# EPICS autosave request: autosave/pu610k.req
#
# List of PVs to autosave.  Assume $(BASE) is the detector base PV,
# $(CHAN) is the channel number/name, and $(IOC) is the IOC base PV.
#
$(BASE):$(CHAN):ENABLE_RBV
$(BASE):$(CHAN):VOLTAGE
$(BASE):$(CHAN):CHARGE_INHIBIT
$(BASE):AUTO_FLASH_ON
$(BASE):FIRE_DELAY
